Staubli VAL3: TrajectoryQueue.pjx

--- TrajectoryQueue.pjx ---
Parameters version=s7.7.2 stackSize=5000 millimeterUnit=true
Program file=clear.pgx
Program file=pop.pgx
Program file=push.pgx
Program file=start.pgx
Program file=stop.pgx
Data file=TrajectoryQueue.dtx
Type name=MotionBuffer path=Disk://MotionBuffer/MotionBuffer.pjx

--- pop.pgx ---
public program pop(MotionBuffer& x_cmd, bool& x_res)
begin
  if (nElems > 0)
    x_cmd = buffer[nPop]
    nElems = nElems - 1
    nPop = nPop + 1
    if (nPop >= size(buffer))
      nPop = 0
    endIf
    x_res = true
  else
    x_res = false
  endIf
end
